PROGRAM Pump
VAR_INPUT
	height : 	LREAL;
	diameter : 	LREAL := 2;
	volume :	LREAL := 25.13;
	fbT1 :		TON;
	FlowValve1 : LREAL := 0;
	FlowValve2 : LREAL := 0;
	FlowSensor1 : LREAL := 0;
	FlowSensor2 : LREAL := 0;
	bValve1Opened			: BOOL;
	bValve2Opened			: BOOL;
	Bottle :	LREAL := 0;
	countFill :	INT := 0;
	// tMove: TIME;
	ClockFill: BOOL := FALSE;
END_VAR
VAR
	ActValve : BOOL := TRUE;
	ActFill : BOOL := TRUE;
	Check_Fill: BOOL := FALSE;
	//ReadyMove1 : BOOL := FALSE;
	//ActMove1: BOOL := FALSE;
END_VAR

//Cylinder Tank: Diameter = 500, Height = 1000
FlowSensor1 := FlowValve1; FlowSensor2 := FlowValve2;
volume := volume + (FlowValve1 - FlowValve2)/100;
height := (4 * volume)/(pi * EXPT(diameter, 2));
IF MAIN.Activate THEN
	IF height >= 9 THEN //Upper level sensor
		FlowValve1 := 0;
		bValve1Opened := FALSE;
	END_IF
	IF height <= 8 THEN //Lower level sensor
		FlowValve1 := 0.251;
		bValve1Opened := TRUE;
	END_IF
	IF NOT ClockFill THEN 
		FlowValve2 := 0.25; 
		bValve2Opened := TRUE;
	ELSE 
		FlowValve2 := 0; 
		bValve2Opened := FALSE;
		JMP label1; //Jump to label1
	END_IF 
	IF countFill >= 1 THEN 
		Seal.enableSeal := TRUE; 
	END_IF
	IF FlowValve2 = 0.25 AND ActFill AND Conveyor.Pos_Bottle1 = 400 THEN
		Bottle := Bottle + FlowValve2/100;
		IF Bottle >= 0.5 AND NOT Check_Fill THEN
			ActFill := FALSE; // Stop Filling
			Check_Fill := TRUE; //Ensure ActFill interrupted once
		END_IF
		IF Bottle >= 0.5 AND Check_Fill THEN
			Bottle := 0;
			countFill := countFill + 1; // Counting Filled Bottle
			// Wait for Transmission
			label1 : fbT1(IN := Check_Fill, PT := T#1S, Q => ActFill);
			ClockFill := TRUE;
			IF ActFill THEN
				fbT1(IN := FALSE);
				Check_Fill := FALSE;
				ClockFill := FALSE;
			END_IF
		END_IF
	END_IF
END_IF

IF NOT MAIN.Activate THEN
	Bottle := 0; height := 8.95;
	FlowValve1 := 0; FlowValve2 := 0;
	countFill := 0; ActFill := TRUE; Check_Fill := FALSE;
	ClockFill := FALSE;
	IF GVL_Fill.bEmergency THEN
		ActValve := FALSE;
	END_IF
END_IF

END_PROGRAM

(* stored: Version 1.1.0.1, ProductVersion 3.1.4024.11
   POU Pump: Id {04fe6544-f8fa-475f-9fc7-5b9abe67aa42}, SpecialFunc None *)
